TYPE U_TICKET_LIST_DATA_OUTPUT :
UNION
  stData              : ST_LIST_NODE_DATA;
  byData   AT %I*     : ARRAY[1..SIZEOF(ST_LIST_NODE_DATA)] OF BYTE;
END_UNION
END_TYPE

(* stored: Version 1.1.0.1
   DUT U_TICKET_LIST_DATA_OUTPUT: Id {dc4393bf-10c6-477b-acc4-8667a49d44b0} *)
